// TIA Portal V18 export
VAR_GLOBAL   // PLC tag table "NGSensor"
   LoadNG3_3 AT %I6400.0 : Bool;
   LoadNG1_4 AT %I6400.1 : Bool;
   LoadNG2_4 AT %I6400.2 : Bool;
   LoadNG3_4 AT %I6400.3 : Bool;
   LoadNG1_5 AT %I6400.4 : Bool;
   LoadNG2_5 AT %I6400.5 : Bool;
   LoadNG3_5 AT %I6400.6 : Bool;
   LoadNG_Spare AT %I6400.7 : Bool;
   LoadNG1_1 AT %I6401.0 : Bool;
   LoadNG2_1 AT %I6401.1 : Bool;
   LoadNG3_1 AT %I6401.2 : Bool;
   LoadNG1_2 AT %I6401.3 : Bool;
   LoadNG2_2 AT %I6401.4 : Bool;
   LoadNG3_2 AT %I6401.5 : Bool;
   LoadNG1_3 AT %I6401.6 : Bool;
   LoadNG2_3 AT %I6401.7 : Bool;
   UnLoadNG3_3 AT %I6500.0 : Bool;
   UnLoadNG1_4 AT %I6500.1 : Bool;
   UnLoadNG2_4 AT %I6500.2 : Bool;
   UnLoadNG3_4 AT %I6500.3 : Bool;
   UnLoadNG1_5 AT %I6500.4 : Bool;
   UnLoadNG2_5 AT %I6500.5 : Bool;
   UnLoadNG3_5 AT %I6500.6 : Bool;
   UnLoadNG_Spare AT %I6500.7 : Bool;
   UnLoadNG1_1 AT %I6501.0 : Bool;
   UnLoadNG2_1 AT %I6501.1 : Bool;
   UnLoadNG3_1 AT %I6501.2 : Bool;
   UnLoadNG1_2 AT %I6501.3 : Bool;
   UnLoadNG2_2 AT %I6501.4 : Bool;
   UnLoadNG3_2 AT %I6501.5 : Bool;
   UnLoadNG1_3 AT %I6501.6 : Bool;
   UnLoadNG2_3 AT %I6501.7 : Bool;
END_VAR
